// TIA Portal V20 export
DATA_BLOCK "AxisDataBackUp_DB"   // DB137
// stored: Access Published, MemoryReserve 100
   VAR
      saveBit : Array[0..20] of Bool;   // DR save button
   END_VAR
   VAR RETAIN
      "emDistance[1]" { ExternalAccessible := 'False'; ExternalVisible := 'False'; ExternalWritable := 'False'} : "LER_typeDistanceInterface";
      "emDistance[2]" { ExternalAccessible := 'False'; ExternalVisible := 'False'; ExternalWritable := 'False'} : "LER_typeDistanceInterface";
      DR1 { ExternalAccessible := 'False'; ExternalVisible := 'False'; ExternalWritable := 'False'} : Struct
         "configuration.setPositions" : Array[0..15] of "LBC_typeAxis64PosSetPosition";
         softcam : "LER_typeSoftCamInterface";
      END_STRUCT;
      DR2 { ExternalAccessible := 'False'; ExternalVisible := 'False'; ExternalWritable := 'False'} : Struct
         "configuration.setPositions" : Array[0..15] of "LBC_typeAxis64PosSetPosition";
         softcam : "LER_typeSoftCamInterface";
      END_STRUCT;
      DR3 { ExternalAccessible := 'False'; ExternalVisible := 'False'; ExternalWritable := 'False'} : Struct
         "configuration.setPositions" : Array[0..15] of "LBC_typeAxis64PosSetPosition";
         softcam : "LER_typeSoftCamInterface";
      END_STRUCT;
      DR4 { ExternalAccessible := 'False'; ExternalVisible := 'False'; ExternalWritable := 'False'} : Struct
         "configuration.setPositions" : Array[0..15] of "LBC_typeAxis64PosSetPosition";
         softcam : "LER_typeSoftCamInterface";
      END_STRUCT;
      DR5 { ExternalAccessible := 'False'; ExternalVisible := 'False'; ExternalWritable := 'False'} : Struct
         "configuration.setPositions" : Array[0..15] of "LBC_typeAxis64PosSetPosition";
         softcam : "LER_typeSoftCamInterface";
      END_STRUCT;
      DR6 { ExternalAccessible := 'False'; ExternalVisible := 'False'; ExternalWritable := 'False'} : Struct
         "configuration.setPositions" : Array[0..15] of "LBC_typeAxis64PosSetPosition";
         softcam : "LER_typeSoftCamInterface";
      END_STRUCT;
      DR7 { ExternalAccessible := 'False'; ExternalVisible := 'False'; ExternalWritable := 'False'} : Struct
         "configuration.setPositions" : Array[0..15] of "LBC_typeAxis64PosSetPosition";
         softcam : "LER_typeSoftCamInterface";
      END_STRUCT;
      DR8 { ExternalAccessible := 'False'; ExternalVisible := 'False'; ExternalWritable := 'False'} : Struct
         "configuration.setPositions" : Array[0..15] of "LBC_typeAxis64PosSetPosition";
         softcam : "LER_typeSoftCamInterface";
      END_STRUCT;
      DR9 { ExternalAccessible := 'False'; ExternalVisible := 'False'; ExternalWritable := 'False'} : Struct
         "configuration.setPositions" : Array[0..15] of "LBC_typeAxis64PosSetPosition";
         softcam : "LER_typeSoftCamInterface";
      END_STRUCT;
      DR10 { ExternalAccessible := 'False'; ExternalVisible := 'False'; ExternalWritable := 'False'} : Struct
         "configuration.setPositions" : Array[0..15] of "LBC_typeAxis64PosSetPosition";
         softcam : "LER_typeSoftCamInterface";
      END_STRUCT;
      DR11 { ExternalAccessible := 'False'; ExternalVisible := 'False'; ExternalWritable := 'False'} : Struct
         "configuration.setPositions" : Array[0..15] of "LBC_typeAxis64PosSetPosition";
         softcam : "LER_typeSoftCamInterface";
      END_STRUCT;
      DR12 { ExternalAccessible := 'False'; ExternalVisible := 'False'; ExternalWritable := 'False'} : Struct
         "configuration.setPositions" : Array[0..15] of "LBC_typeAxis64PosSetPosition";
         softcam : "LER_typeSoftCamInterface";
      END_STRUCT;
      DR13 { ExternalAccessible := 'False'; ExternalVisible := 'False'; ExternalWritable := 'False'} : Struct
         "configuration.setPositions" : Array[0..15] of "LBC_typeAxis64PosSetPosition";
         softcam : "LER_typeSoftCamInterface";
      END_STRUCT;
      DR14 { ExternalAccessible := 'False'; ExternalVisible := 'False'; ExternalWritable := 'False'} : Struct
         "configuration.setPositions" : Array[0..15] of "LBC_typeAxis64PosSetPosition";
         softcam : "LER_typeSoftCamInterface";
      END_STRUCT;
      DR15 { ExternalAccessible := 'False'; ExternalVisible := 'False'; ExternalWritable := 'False'} : Struct
         "configuration.setPositions" : Array[0..15] of "LBC_typeAxis64PosSetPosition";
         softcam : "LER_typeSoftCamInterface";
      END_STRUCT;
      DR16 { ExternalAccessible := 'False'; ExternalVisible := 'False'; ExternalWritable := 'False'} : Struct
         "configuration.setPositions" : Array[0..15] of "LBC_typeAxis64PosSetPosition";
         softcam : "LER_typeSoftCamInterface";
      END_STRUCT;
      DR17 { ExternalAccessible := 'False'; ExternalVisible := 'False'; ExternalWritable := 'False'} : Struct
         "configuration.setPositions" : Array[0..15] of "LBC_typeAxis64PosSetPosition";
         softcam : "LER_typeSoftCamInterface";
      END_STRUCT;
      DR18 { ExternalAccessible := 'False'; ExternalVisible := 'False'; ExternalWritable := 'False'} : Struct
         "configuration.setPositions" : Array[0..15] of "LBC_typeAxis64PosSetPosition";
         softcam : "LER_typeSoftCamInterface";
      END_STRUCT;
      DR19 { ExternalAccessible := 'False'; ExternalVisible := 'False'; ExternalWritable := 'False'} : Struct
         "configuration.setPositions" : Array[0..15] of "LBC_typeAxis64PosSetPosition";
         softcam : "LER_typeSoftCamInterface";
      END_STRUCT;
      DR20 { ExternalAccessible := 'False'; ExternalVisible := 'False'; ExternalWritable := 'False'} : Struct
         "configuration.setPositions" : Array[0..15] of "LBC_typeAxis64PosSetPosition";
         softcam : "LER_typeSoftCamInterface";
      END_STRUCT;
   END_VAR
BEGIN
END_DATA_BLOCK
